FUNCTION_BLOCK FB_Handle_Emergency
VAR_INPUT
    execute: 				BOOL;
END_VAR
VAR_OUTPUT
    busy: 					BOOL;
    done: 					BOOL;
END_VAR
VAR
    state: 					INT := 0;
    tonDelay: 				TON;
	allActionsComplete:		BOOL;
END_VAR

IF NOT execute THEN
    state := 0;
    busy := FALSE;
    done := FALSE;
    tonDelay(IN := FALSE);
    RETURN;
END_IF

//trigger EL!
busy := TRUE;
CASE state OF
    0:  GVL_FSM.open_SDC := TRUE;
        GVL_FSM.engage_brakes := TRUE;
        GVL_Prop.propulsion_enable := FALSE;
        GVL_Levi.levitation_active := FALSE;
        GVL_PT.emergency_shutdown := TRUE;
        state := 1;
        
    1:  allActionsComplete := 
            NOT GVL_FSM.sdc_closed AND
            GVL_FSM.brakes_engaged AND
            NOT GVL_Prop.propulsion_active AND
            NOT GVL_Levi.levitation_active;
        
        IF allActionsComplete THEN
            state := 2;
        END_IF
        
    2:	tonDelay(IN := TRUE, PT := T#200MS);
        IF tonDelay.Q THEN
            busy := FALSE;
            done := TRUE;
        END_IF
END_CASE

END_FUNCTION_BLOCK

(* stored: Version 1.1.0.1
   POU FB_Handle_Emergency: Id {5e0fb178-c06f-42de-8ba0-d84d3592dd6b}, SpecialFunc None *)
